TYPE PowerOfService_Struct :
STRUCT
	InertiaEmulationP_Service : REAL;
	FrequencyRegulationP_Service : REAL;
	ModalFreqAttP_Service : REAL;
	VoltageRegulationQ_Service : REAL;
END_STRUCT
END_TYPE

(* stored: Version 1.1.0.1, ProductVersion 3.1.4022.12
   DUT PowerOfService_Struct: Id {217b7c86-f5a8-4942-9954-01d68d2d9f0b} *)
